FUNCTION_BLOCK SS3_ps_PnP (* Composite FB wrapping other FBs *)
  (* Standard: 61499-2 *)
  (* Version 1.0, 2025-08-24, PS_Transformer_for_Unknown *)
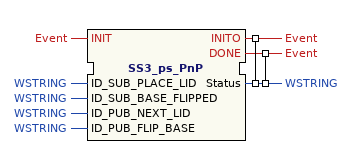
  EVENT_INPUT
    INIT; (* Initialization Request *)
  END_EVENT
  EVENT_OUTPUT
    INITO WITH Status; (* Initialization Confirm *)
    DONE WITH Status; (* Execution Confirmation *)
  END_EVENT
  VAR_INPUT
    ID_SUB_PLACE_LID : WSTRING;
    ID_SUB_BASE_FLIPPED : WSTRING;
    ID_PUB_NEXT_LID : WSTRING;
    ID_PUB_FLIP_BASE : WSTRING;
  END_VAR
  VAR_OUTPUT
    Status : WSTRING; (* Output event qualifier *)
  END_VAR
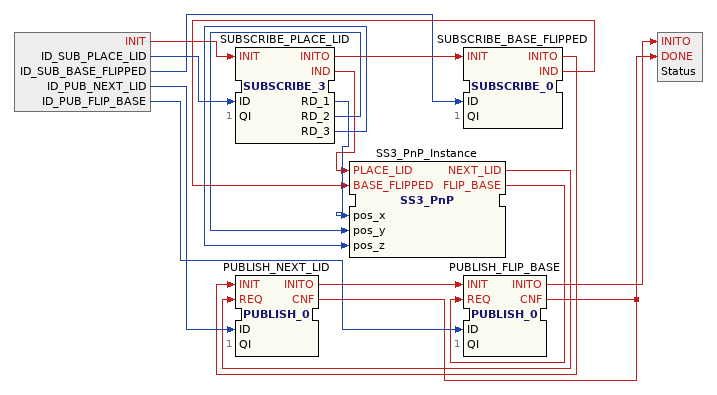
  FBS
    SS3_PnP_Instance : SS3_PnP;
    SUBSCRIBE_PLACE_LID : SUBSCRIBE_3(QI := 1);
    SUBSCRIBE_BASE_FLIPPED : SUBSCRIBE_0(QI := 1);
    PUBLISH_NEXT_LID : PUBLISH_0(QI := 1);
    PUBLISH_FLIP_BASE : PUBLISH_0(QI := 1);
  END_FBS
  EVENT_CONNECTIONS
    INIT TO SUBSCRIBE_PLACE_LID.INIT;
    SUBSCRIBE_PLACE_LID.INITO TO SUBSCRIBE_BASE_FLIPPED.INIT;
    SUBSCRIBE_BASE_FLIPPED.INITO TO PUBLISH_NEXT_LID.INIT;
    PUBLISH_NEXT_LID.INITO TO PUBLISH_FLIP_BASE.INIT;
    PUBLISH_FLIP_BASE.INITO TO INITO;
    SUBSCRIBE_PLACE_LID.IND TO SS3_PnP_Instance.PLACE_LID;
    SUBSCRIBE_BASE_FLIPPED.IND TO SS3_PnP_Instance.BASE_FLIPPED;
    SS3_PnP_Instance.NEXT_LID TO PUBLISH_NEXT_LID.REQ;
    SS3_PnP_Instance.FLIP_BASE TO PUBLISH_FLIP_BASE.REQ;
    PUBLISH_NEXT_LID.CNF TO DONE;
    PUBLISH_FLIP_BASE.CNF TO DONE;
  END_CONNECTIONS
  DATA_CONNECTIONS
    ID_SUB_PLACE_LID TO SUBSCRIBE_PLACE_LID.ID;
    ID_SUB_BASE_FLIPPED TO SUBSCRIBE_BASE_FLIPPED.ID;
    ID_PUB_NEXT_LID TO PUBLISH_NEXT_LID.ID;
    ID_PUB_FLIP_BASE TO PUBLISH_FLIP_BASE.ID;
    SUBSCRIBE_PLACE_LID.RD_1 TO SS3_PnP_Instance.pos_x;
    SUBSCRIBE_PLACE_LID.RD_2 TO SS3_PnP_Instance.pos_y;
    SUBSCRIBE_PLACE_LID.RD_3 TO SS3_PnP_Instance.pos_z;
  END_CONNECTIONS
END_FUNCTION_BLOCK
